{attribute 'analysis' := '-33'}
PROGRAM INTERNAL PRG_IssuesTests
VAR
{IF defined (UNIT_TEST)}
	fbIssue4Tests : FB_Issue4Tests;
{END_IF}
END_VAR

END_PROGRAM

(* stored: Version 1.1.0.1
   POU PRG_IssuesTests: Id {f025cc18-9990-4034-a080-14ae578f3eed}, SpecialFunc None *)
